(* Logix 5000 project; controller RetoFinal Emulate 5570 rev 30.12; software revision 30.00 *)

TASK MainTask (continuous, watchdog 500 ms) : MainProgram

MODULES
   Local : Emulate 5570 (ICP 2, rev 30.12)
END_MODULES

VAR_GLOBAL   (* controller tags *)
   CajaLlego2 : BOOL;
   CajaPaso2 : BOOL;
   CajaPaso3 : BOOL;
   CondicionInicial : BOOL;
   ControlBarrera : BOOL;
   CounterCajas : COUNTER := (PRE := 1);
   GD_A00 : BOOL;
   GD_A00B : BOOL;
   GD_A01 : BOOL;
   GD_A01B : BOOL;
   GD_A10 : BOOL;
   GD_A10B : BOOL;
   GD_A11 : BOOL;
   GD_A11B : BOOL;
   GD_B0 : BOOL := 1;
   GD_B1 : BOOL;
   GD_B1B : BOOL;
   GD_B2 : BOOL;
   GD_B2B : BOOL;
   GD_B3 : BOOL;
   GD_B3B : BOOL;
   GD_B3C : BOOL;
   GD_B3D : BOOL;
   GD_B4 : BOOL := 1;
   GD_B4B : BOOL := 1;
   GD_B5 : BOOL := 1;
   GD_IN_1 : BOOL;
   GD_IN_2 : BOOL;
   GD_IN_3 : BOOL;
   GD_IN_5 : BOOL;
   GD_IN_6 : BOOL;
   GD_OUT_0 : BOOL;
   GD_OUT_4 : BOOL;
   GD_OUT_5 : BOOL;
   GD_P0 : INT;
   GD_P1 : INT;
   GD_P2 : INT;
   GD_P3 : INT;
   GD_P4 : INT;
   GD_P5 : INT;
   GD_P6 : INT;
   GD_P7 : INT;
   GD_P8 : INT;
   GD_P9 : INT;
   GD_R00 : BOOL := 1;
   GD_R00B : BOOL := 1;
   GD_R01 : BOOL;
   GD_R01B : BOOL;
   GD_R10 : BOOL := 1;
   GD_R11 : BOOL;
   GD_S0 : BOOL;
   GD_S1 : BOOL;
   GD_S10 : BOOL;
   GD_S11 : BOOL;
   GD_S2 : BOOL;
   GD_S3 : BOOL;
   GD_S4 : BOOL;
   GD_S5 : BOOL;
   GD_S6 : BOOL;
   GD_S7 : BOOL;
   GD_S8 : BOOL;
   GD_S9 : BOOL;
   IoT_A00 : BOOL;
   IoT_A01 : BOOL;
   IoT_A10 : BOOL;
   IoT_A11 : BOOL;
   IoT_B0 : BOOL := 1;
   IoT_B1 : BOOL;
   IoT_B2 : BOOL;
   IoT_B3 : BOOL;
   IoT_B4 : BOOL := 1;
   IoT_B5 : BOOL := 1;
   IoT_P0 : INT;
   IoT_P1 : INT;
   IoT_P2 : INT;
   IoT_P3 : INT;
   IoT_P4 : INT;
   IoT_P5 : INT;
   IoT_P6 : INT;
   IoT_P7 : INT;
   IoT_P8 : INT;
   IoT_P9 : INT;
   IoT_R00 : BOOL := 1;
   IoT_R01 : BOOL;
   IoT_R10 : BOOL := 1;
   IoT_R11 : BOOL;
   IoT_S0 : BOOL;
   IoT_S1 : BOOL;
   IoT_S2 : BOOL;
   IoT_S3 : BOOL;
   IoT_S4 : BOOL;
   IoT_S5 : BOOL;
   IoT_S6 : BOOL;
   IoT_S7 : BOOL;
   IoT_S8 : BOOL;
   IoT_S9 : BOOL;
   IoT_Tipo : BOOL;
   Sensor2Down : BOOL;
   Sensor2Up : BOOL;
   Sensor3Up : BOOL;
   T1 : TIMER := (PRE := 1000);
END_VAR

PROGRAM MainProgram   (* main routine MainRoutine *)
VAR
   A00 : BOOL;
   A01 : BOOL;
   A10 : BOOL;
   A11 : BOOL;
   AcomodadorSalidaD : BOOL;
   AcomodadorSalidaL : BOOL;
   B0 : BOOL := 1;
   B1 : BOOL;
   B2 : BOOL;
   B3 : BOOL;
   B4 : BOOL := 1;
   B5 : BOOL := 1;
   C1 : COUNTER := (PRE := 2);
   C2 : COUNTER := (PRE := 2);
   CAJAS : DINT;
   CambioTipo : BOOL;
   E00 : BOOL := 1;
   E001 : BOOL := 1;
   E002 : BOOL;
   E01 : BOOL;
   E1 : BOOL := 1;
   E11 : BOOL := 1;
   E12 : BOOL;
   E2 : BOOL;
   E21 : BOOL;
   E22 : BOOL;
   E23 : BOOL;
   E24 : BOOL;
   E25 : BOOL;
   E26 : BOOL;
   E3 : BOOL := 1;
   F : BOOL;
   F1 : BOOL;
   FIN : BOOL := 1;
   FINE2 : BOOL;
   FINE3 : BOOL;
   GD_IN_4 : BOOL;
   M : BOOL;
   M1 : BOOL;
   P0 : INT;
   P1 : INT;
   P2 : INT;
   P3 : INT;
   P4 : INT;
   P5 : INT;
   P6 : INT;
   P7 : INT;
   P8 : INT;
   P9 : INT;
   R00 : BOOL := 1;
   R01 : BOOL;
   R10 : BOOL := 1;
   R11 : BOOL;
   S0 : BOOL;
   S0D : BOOL;
   S0Dw : BOOL;
   S0U : BOOL;
   S0Up : BOOL;
   S1 : BOOL;
   S10 : BOOL;
   S10D : BOOL;
   S10Dw : BOOL;
   S10U : BOOL;
   S10Up : BOOL;
   S11 : BOOL;
   S11D : BOOL;
   S11Dw : BOOL;
   S11U : BOOL;
   S11Up : BOOL;
   S1D : BOOL;
   S1Dw : BOOL;
   S1U : BOOL;
   S1Up : BOOL;
   S2 : BOOL;
   S2D : BOOL;
   S2Dw : BOOL;
   S2U : BOOL;
   S2Up : BOOL;
   S3 : BOOL;
   S3D : BOOL;
   S3Dw : BOOL;
   S3U : BOOL;
   S3Up : BOOL;
   S4 : BOOL;
   S4D : BOOL;
   S4Dw : BOOL;
   S4U : BOOL;
   S4Up : BOOL;
   S5 : BOOL;
   S5D : BOOL;
   S5Dw : BOOL;
   S5U : BOOL;
   S5Up : BOOL;
   S6 : BOOL;
   S6D : BOOL;
   S6Dw : BOOL;
   S6U : BOOL;
   S6Up : BOOL;
   S7 : BOOL;
   S7D : BOOL;
   S7Dw : BOOL;
   S7U : BOOL;
   S7Up : BOOL;
   S8 : BOOL;
   S8D : BOOL;
   S8Dw : BOOL;
   S8U : BOOL;
   S8Up : BOOL;
   S9 : BOOL;
   S9D : BOOL;
   S9Dw : BOOL;
   S9U : BOOL;
   S9Up : BOOL;
   SistemaActivo : BOOL := 1;
   TimerBarrera : TIMER := (PRE := 500);
   Tipo : BOOL;
   TipoD : BOOL;
   TipoDw : BOOL;
   TipoU : BOOL;
   TipoUp : BOOL;
END_VAR

ROUTINE A   (* ladder *)
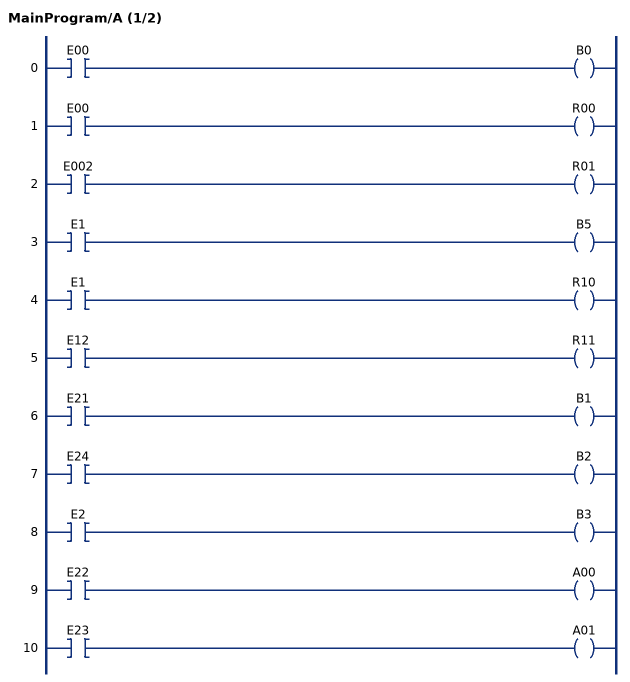
   0: XIC(E00)OTE(B0);
   1: XIC(E00)OTE(R00);
   2: XIC(E002)OTE(R01);
   3: XIC(E1)OTE(B5);
   4: XIC(E1)OTE(R10);
   5: XIC(E12)OTE(R11);
   6: XIC(E21)OTE(B1);
   7: XIC(E24)OTE(B2);
   8: XIC(E2)OTE(B3);
   9: XIC(E22)OTE(A00);
   10: XIC(E23)OTE(A01);
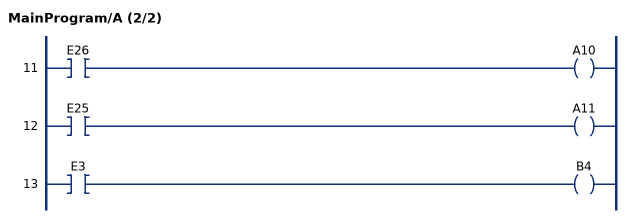
   11: XIC(E26)OTE(A10);
   12: XIC(E25)OTE(A11);
   13: XIC(E3)OTE(B4);
END_ROUTINE

ROUTINE Buffer   (* ladder *)
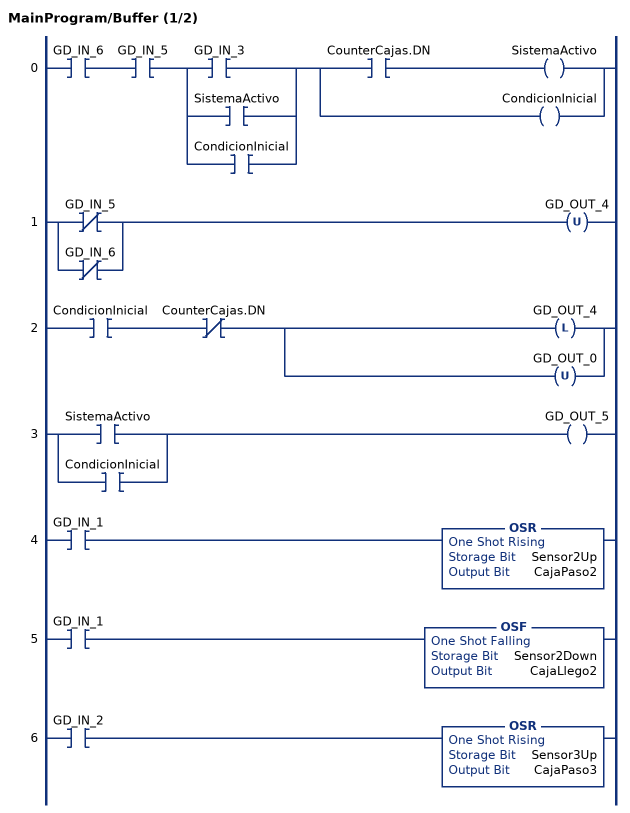
   0: XIC(GD_IN_6)XIC(GD_IN_5)[XIC(GD_IN_3) ,[XIC(SistemaActivo) ,XIC(CondicionInicial) ] ][XIC(CounterCajas.DN) OTE(SistemaActivo) ,OTE(CondicionInicial) ];
   1: [XIO(GD_IN_5) ,XIO(GD_IN_6) ]OTU(GD_OUT_4);
   2: XIC(CondicionInicial)XIO(CounterCajas.DN)[OTL(GD_OUT_4) ,OTU(GD_OUT_0) ];
   3: [XIC(SistemaActivo) ,XIC(CondicionInicial) ]OTE(GD_OUT_5);
   4: XIC(GD_IN_1)OSR(Sensor2Up,CajaPaso2);
   5: XIC(GD_IN_1)OSF(Sensor2Down,CajaLlego2);
   6: XIC(GD_IN_2)OSR(Sensor3Up,CajaPaso3);
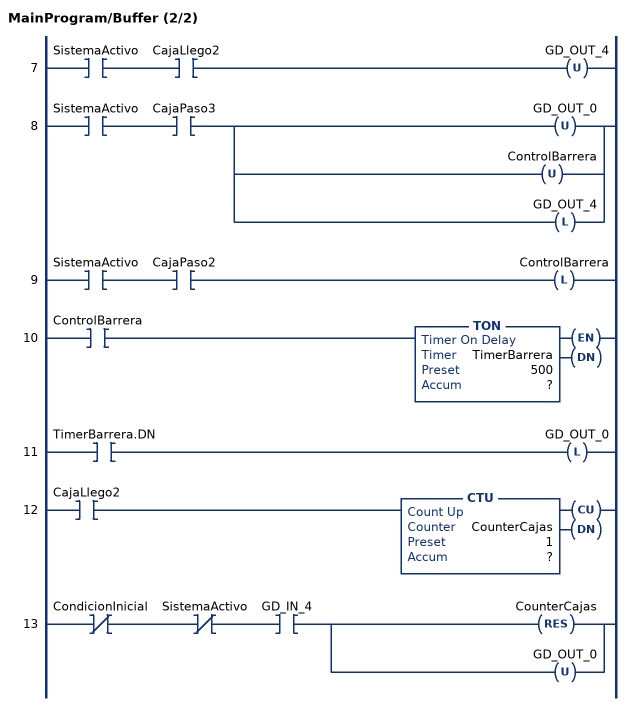
   7: XIC(SistemaActivo)XIC(CajaLlego2)OTU(GD_OUT_4);
   8: XIC(SistemaActivo)XIC(CajaPaso3)[OTU(GD_OUT_0) ,[OTU(ControlBarrera) ,OTL(GD_OUT_4) ] ];
   9: XIC(SistemaActivo)XIC(CajaPaso2)OTL(ControlBarrera);
   10: XIC(ControlBarrera)TON(TimerBarrera,?,?);
   11: XIC(TimerBarrera.DN)OTL(GD_OUT_0);
   12: XIC(CajaLlego2)CTU(CounterCajas,?,?);
   13: XIO(CondicionInicial)XIO(SistemaActivo)XIC(GD_IN_4)[RES(CounterCajas) ,OTU(GD_OUT_0) ];
END_ROUTINE

ROUTINE C   (* ladder *)
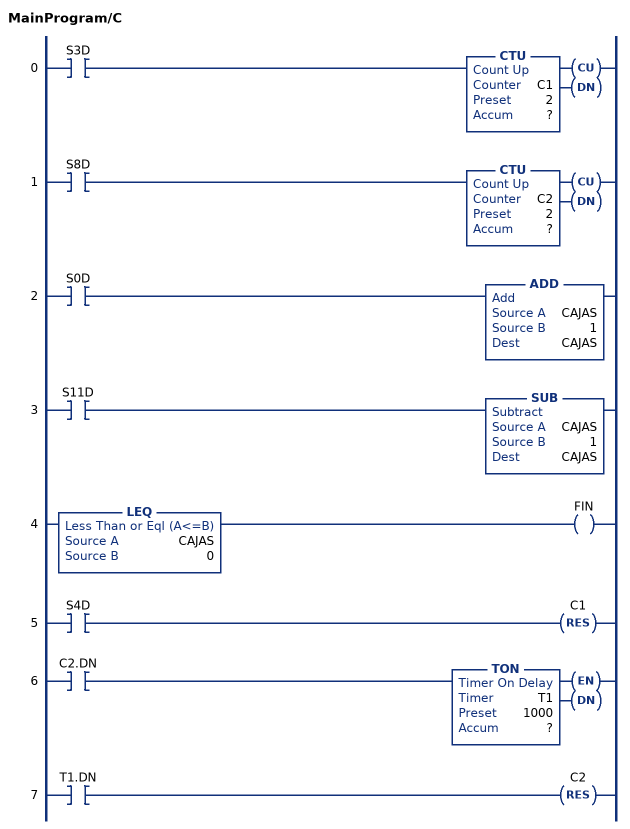
   0: XIC(S3D)CTU(C1,?,?);
   1: XIC(S8D)CTU(C2,?,?);
   2: XIC(S0D)ADD(CAJAS,1,CAJAS);
   3: XIC(S11D)SUB(CAJAS,1,CAJAS);
   4: LEQ(CAJAS,0)OTE(FIN);
   5: XIC(S4D)RES(C1);
   6: XIC(C2.DN)TON(T1,?,?);
   7: XIC(T1.DN)RES(C2);
END_ROUTINE

ROUTINE E   (* ladder *)
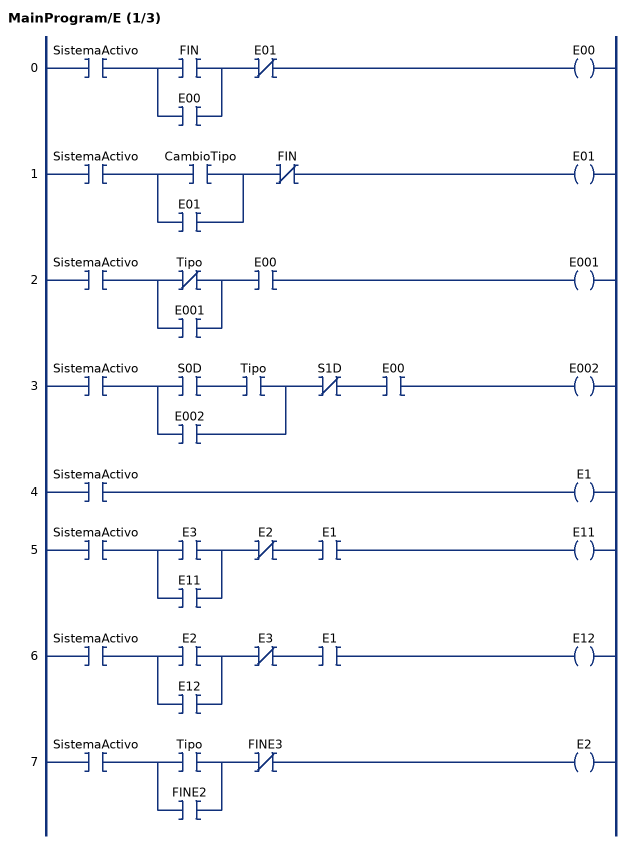
   0: XIC(SistemaActivo)[XIC(FIN) ,XIC(E00) ]XIO(E01)OTE(E00);
   1: XIC(SistemaActivo)[XIC(CambioTipo) ,XIC(E01) ]XIO(FIN)OTE(E01);
   2: XIC(SistemaActivo)[XIO(Tipo) ,XIC(E001) ]XIC(E00)OTE(E001);
   3: XIC(SistemaActivo)[XIC(S0D) XIC(Tipo) ,XIC(E002) ]XIO(S1D)XIC(E00)OTE(E002);
   4: XIC(SistemaActivo)OTE(E1);
   5: XIC(SistemaActivo)[XIC(E3) ,XIC(E11) ]XIO(E2)XIC(E1)OTE(E11);
   6: XIC(SistemaActivo)[XIC(E2) ,XIC(E12) ]XIO(E3)XIC(E1)OTE(E12);
   7: XIC(SistemaActivo)[XIC(Tipo) ,XIC(FINE2) ]XIO(FINE3)OTE(E2);
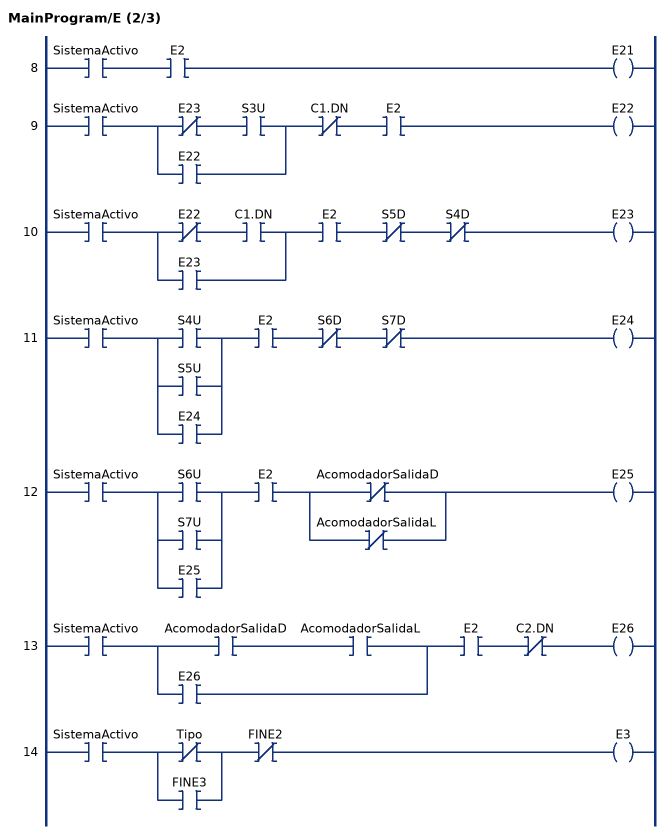
   8: XIC(SistemaActivo)XIC(E2)OTE(E21);
   9: XIC(SistemaActivo)[XIO(E23) XIC(S3U) ,XIC(E22) ]XIO(C1.DN)XIC(E2)OTE(E22);
   10: XIC(SistemaActivo)[XIO(E22) XIC(C1.DN) ,XIC(E23) ]XIC(E2)XIO(S5D)XIO(S4D)OTE(E23);
   11: XIC(SistemaActivo)[[XIC(S4U) ,XIC(S5U) ] ,XIC(E24) ]XIC(E2)XIO(S6D)XIO(S7D)OTE(E24);
   12: XIC(SistemaActivo)[[XIC(S6U) ,XIC(S7U) ] ,XIC(E25) ]XIC(E2)[XIO(AcomodadorSalidaD) ,XIO(AcomodadorSalidaL) ]OTE(E25);
   13: XIC(SistemaActivo)[XIC(AcomodadorSalidaD) XIC(AcomodadorSalidaL) ,XIC(E26) ]XIC(E2)XIO(C2.DN)OTE(E26);
   14: XIC(SistemaActivo)[XIO(Tipo) ,XIC(FINE3) ]XIO(FINE2)OTE(E3);
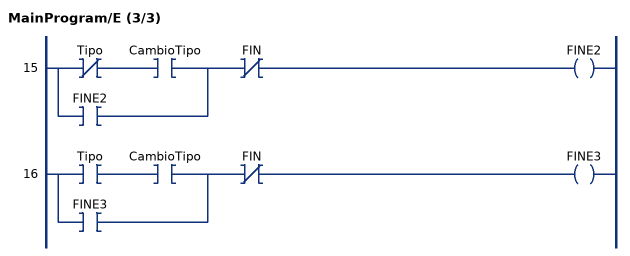
   15: [XIO(Tipo) XIC(CambioTipo) ,XIC(FINE2) ]XIO(FIN)OTE(FINE2);
   16: [XIC(Tipo) XIC(CambioTipo) ,XIC(FINE3) ]XIO(FIN)OTE(FINE3);
END_ROUTINE

ROUTINE GD   (* ladder *)
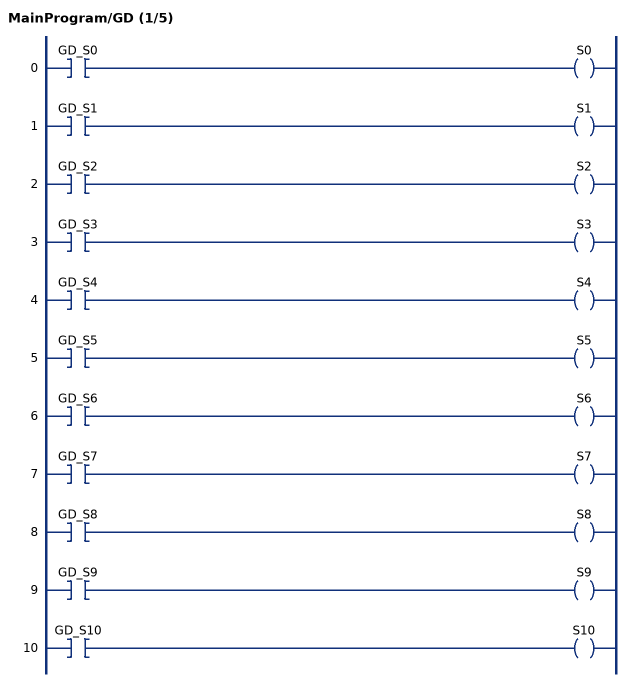
   0: XIC(GD_S0)OTE(S0);
   1: XIC(GD_S1)OTE(S1);
   2: XIC(GD_S2)OTE(S2);
   3: XIC(GD_S3)OTE(S3);
   4: XIC(GD_S4)OTE(S4);
   5: XIC(GD_S5)OTE(S5);
   6: XIC(GD_S6)OTE(S6);
   7: XIC(GD_S7)OTE(S7);
   8: XIC(GD_S8)OTE(S8);
   9: XIC(GD_S9)OTE(S9);
   10: XIC(GD_S10)OTE(S10);
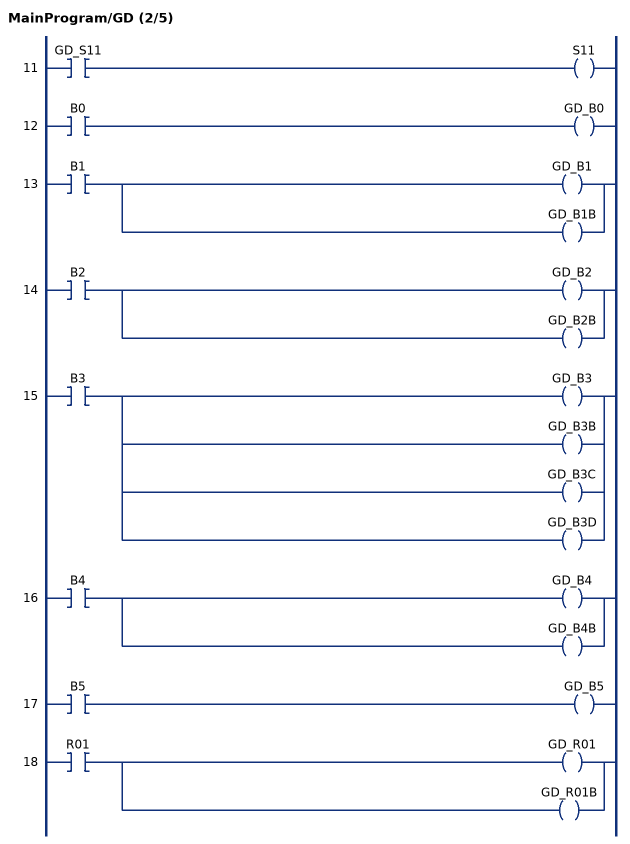
   11: XIC(GD_S11)OTE(S11);
   12: XIC(B0)OTE(GD_B0);
   13: XIC(B1)[OTE(GD_B1) ,OTE(GD_B1B) ];
   14: XIC(B2)[OTE(GD_B2) ,OTE(GD_B2B) ];
   15: XIC(B3)[OTE(GD_B3) ,[OTE(GD_B3B) ,[OTE(GD_B3C) ,OTE(GD_B3D) ] ] ];
   16: XIC(B4)[OTE(GD_B4) ,OTE(GD_B4B) ];
   17: XIC(B5)OTE(GD_B5);
   18: XIC(R01)[OTE(GD_R01) ,OTE(GD_R01B) ];
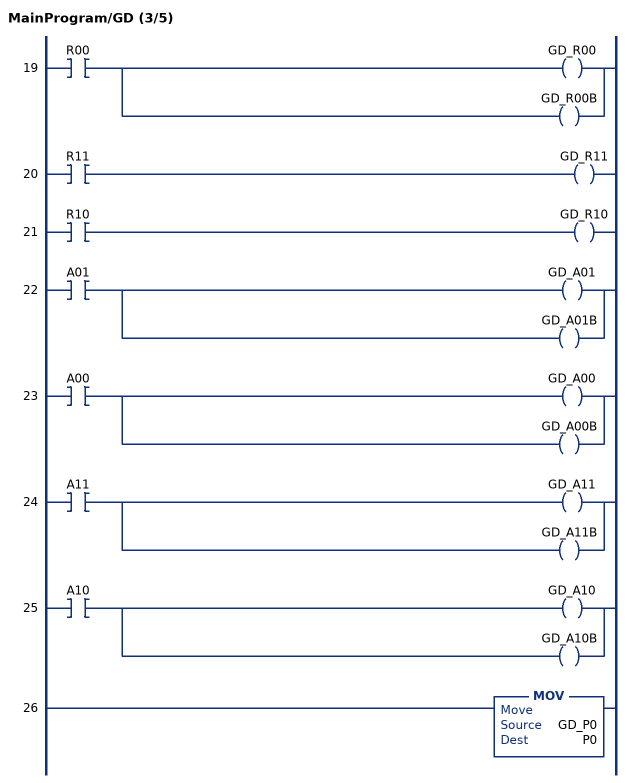
   19: XIC(R00)[OTE(GD_R00) ,OTE(GD_R00B) ];
   20: XIC(R11)OTE(GD_R11);
   21: XIC(R10)OTE(GD_R10);
   22: XIC(A01)[OTE(GD_A01) ,OTE(GD_A01B) ];
   23: XIC(A00)[OTE(GD_A00) ,OTE(GD_A00B) ];
   24: XIC(A11)[OTE(GD_A11) ,OTE(GD_A11B) ];
   25: XIC(A10)[OTE(GD_A10) ,OTE(GD_A10B) ];
   26: MOV(GD_P0,P0);
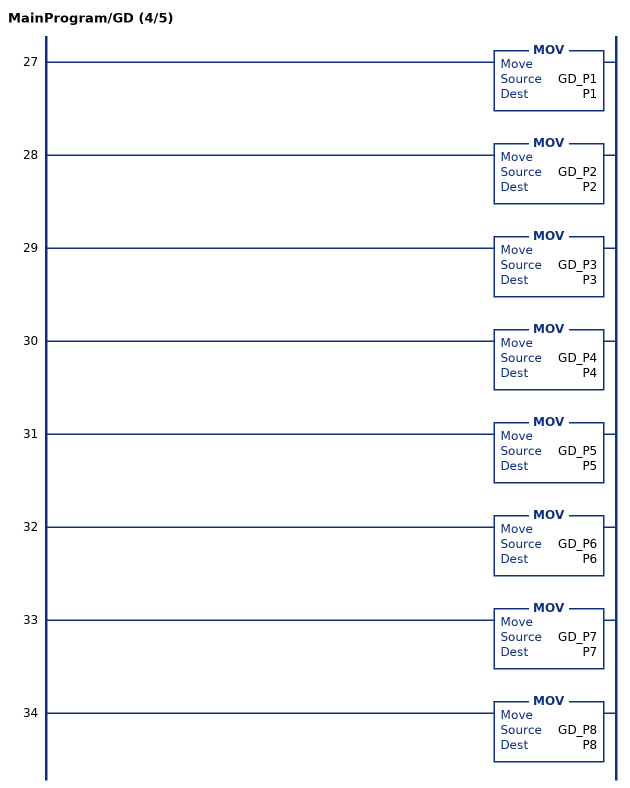
   27: MOV(GD_P1,P1);
   28: MOV(GD_P2,P2);
   29: MOV(GD_P3,P3);
   30: MOV(GD_P4,P4);
   31: MOV(GD_P5,P5);
   32: MOV(GD_P6,P6);
   33: MOV(GD_P7,P7);
   34: MOV(GD_P8,P8);
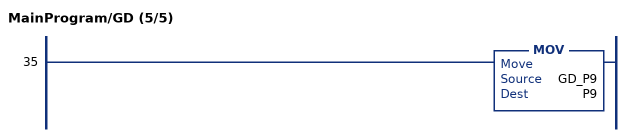
   35: MOV(GD_P9,P9);
END_ROUTINE

ROUTINE IoT   (* ladder *)
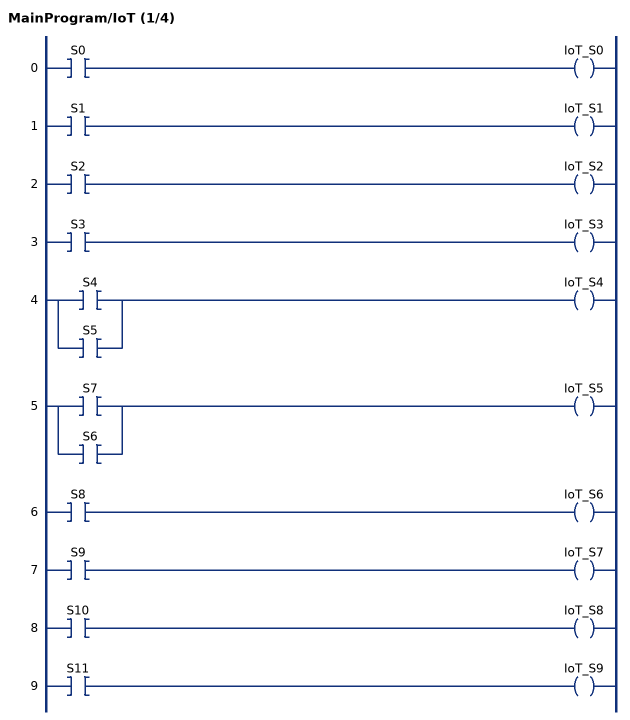
   0: XIC(S0)OTE(IoT_S0);
   1: XIC(S1)OTE(IoT_S1);
   2: XIC(S2)OTE(IoT_S2);
   3: XIC(S3)OTE(IoT_S3);
   4: [XIC(S4) ,XIC(S5) ]OTE(IoT_S4);
   5: [XIC(S7) ,XIC(S6) ]OTE(IoT_S5);
   6: XIC(S8)OTE(IoT_S6);
   7: XIC(S9)OTE(IoT_S7);
   8: XIC(S10)OTE(IoT_S8);
   9: XIC(S11)OTE(IoT_S9);
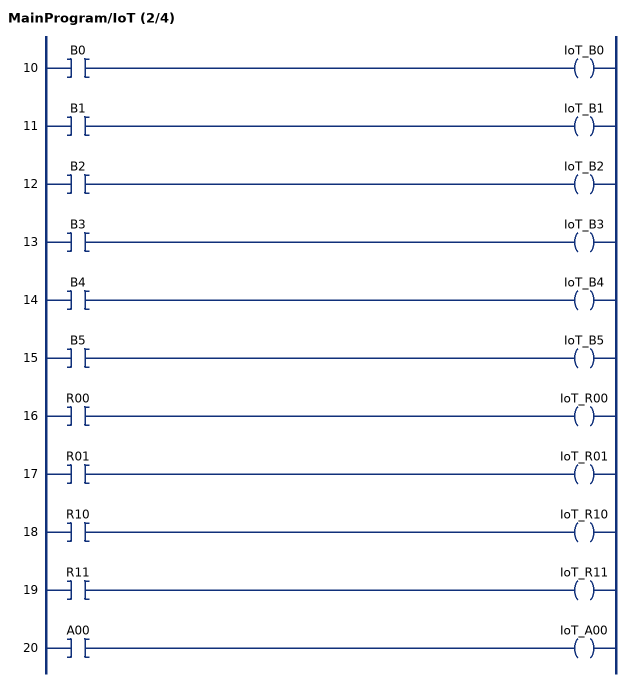
   10: XIC(B0)OTE(IoT_B0);
   11: XIC(B1)OTE(IoT_B1);
   12: XIC(B2)OTE(IoT_B2);
   13: XIC(B3)OTE(IoT_B3);
   14: XIC(B4)OTE(IoT_B4);
   15: XIC(B5)OTE(IoT_B5);
   16: XIC(R00)OTE(IoT_R00);
   17: XIC(R01)OTE(IoT_R01);
   18: XIC(R10)OTE(IoT_R10);
   19: XIC(R11)OTE(IoT_R11);
   20: XIC(A00)OTE(IoT_A00);
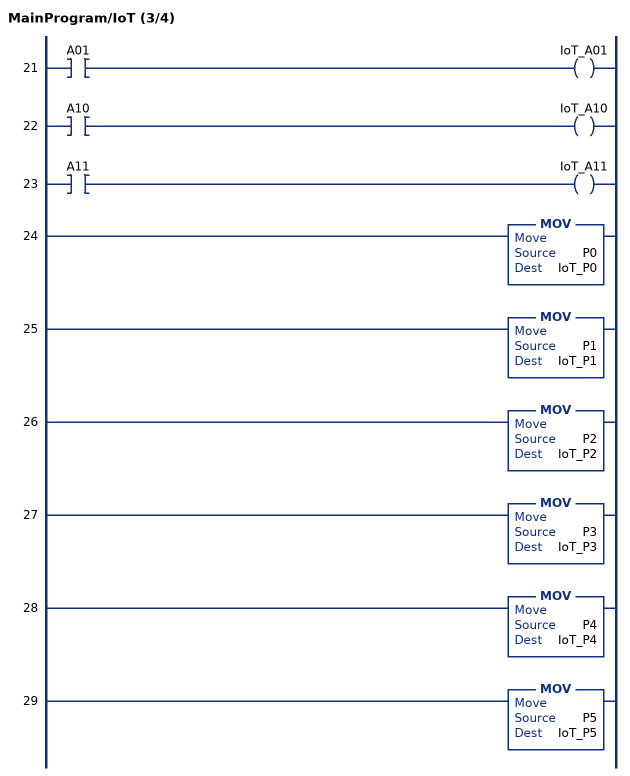
   21: XIC(A01)OTE(IoT_A01);
   22: XIC(A10)OTE(IoT_A10);
   23: XIC(A11)OTE(IoT_A11);
   24: MOV(P0,IoT_P0);
   25: MOV(P1,IoT_P1);
   26: MOV(P2,IoT_P2);
   27: MOV(P3,IoT_P3);
   28: MOV(P4,IoT_P4);
   29: MOV(P5,IoT_P5);
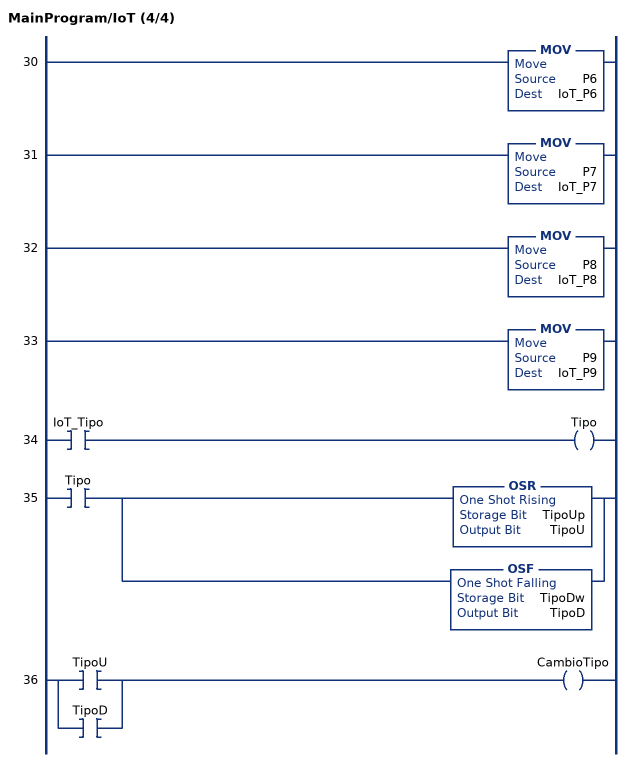
   30: MOV(P6,IoT_P6);
   31: MOV(P7,IoT_P7);
   32: MOV(P8,IoT_P8);
   33: MOV(P9,IoT_P9);
   34: XIC(IoT_Tipo)OTE(Tipo);
   35: XIC(Tipo)[OSR(TipoUp,TipoU) ,OSF(TipoDw,TipoD) ];
   36: [XIC(TipoU) ,XIC(TipoD) ]OTE(CambioTipo);
END_ROUTINE

ROUTINE MainRoutine   (* ladder *)
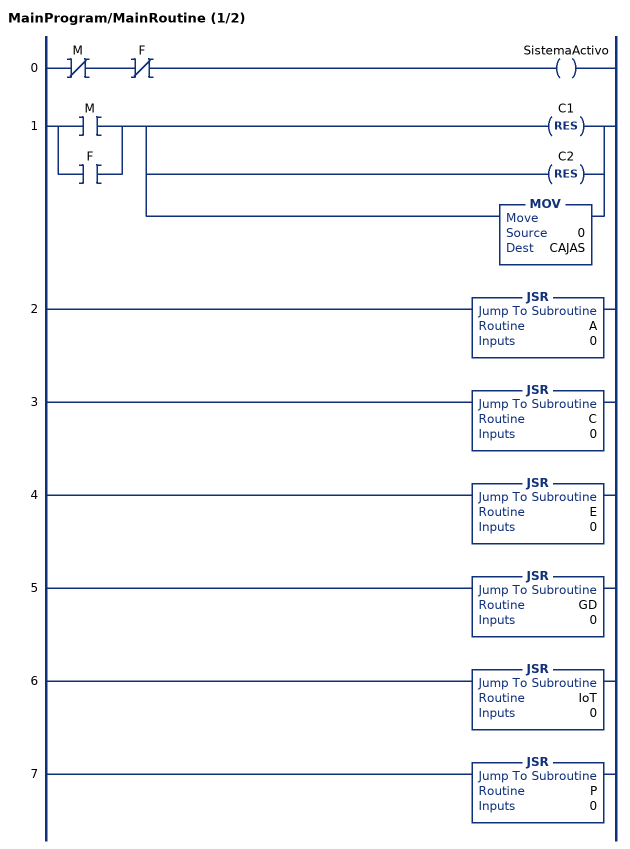
   0: XIO(M)XIO(F)OTE(SistemaActivo);
   1: [XIC(M) ,XIC(F) ][RES(C1) ,[RES(C2) ,MOV(0,CAJAS) ] ];
   2: JSR(A,0);
   3: JSR(C,0);
   4: JSR(E,0);
   5: JSR(GD,0);
   6: JSR(IoT,0);
   7: JSR(P,0);
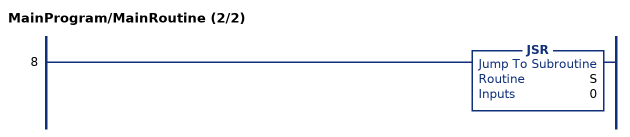
   8: JSR(S,0);
END_ROUTINE

ROUTINE P   (* ladder *)
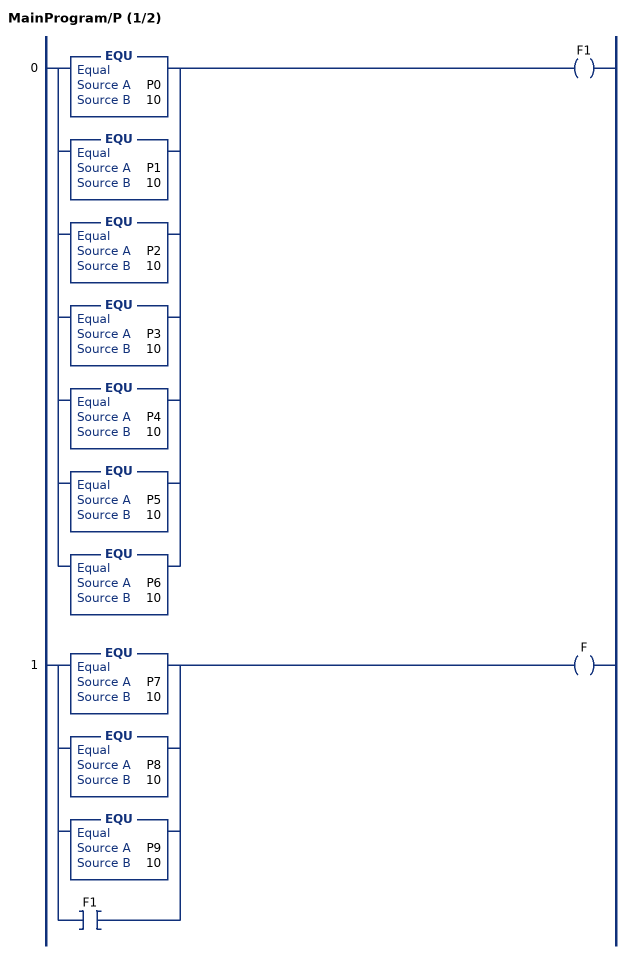
   0: [EQU(P0,10) ,[EQU(P1,10) ,[EQU(P2,10) ,[EQU(P3,10) ,[EQU(P4,10) ,[EQU(P5,10) ,EQU(P6,10) ] ] ] ] ] ]OTE(F1);
   1: [EQU(P7,10) ,[EQU(P8,10) ,[EQU(P9,10) ,XIC(F1) ] ] ]OTE(F);
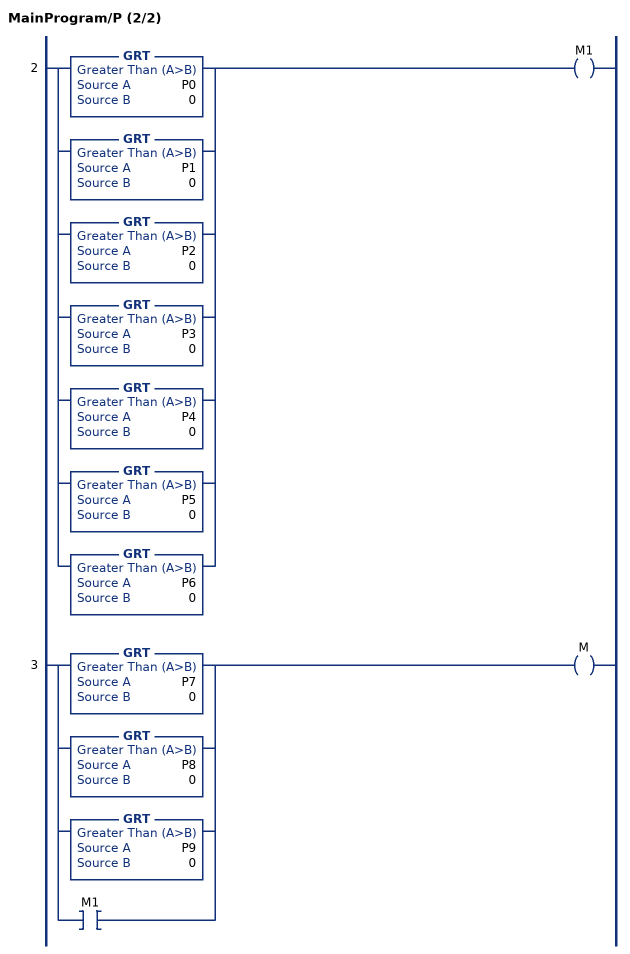
   2: [GRT(P0,0) ,[GRT(P1,0) ,[GRT(P2,0) ,[GRT(P3,0) ,[GRT(P4,0) ,[GRT(P5,0) ,GRT(P6,0) ] ] ] ] ] ]OTE(M1);
   3: [GRT(P7,0) ,[GRT(P8,0) ,[GRT(P9,0) ,XIC(M1) ] ] ]OTE(M);
END_ROUTINE

ROUTINE S   (* ladder *)
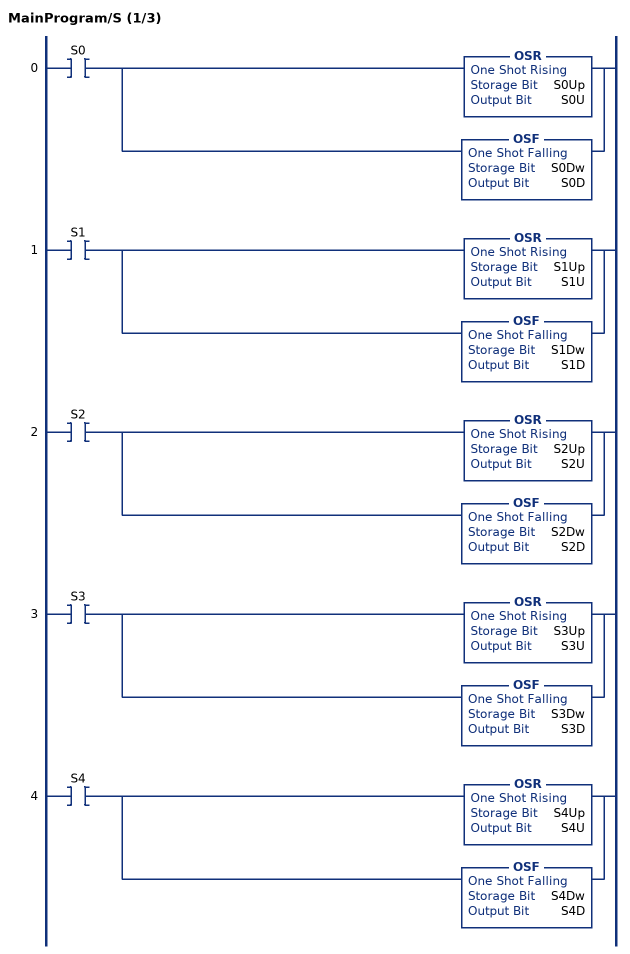
   0: XIC(S0)[OSR(S0Up,S0U) ,OSF(S0Dw,S0D) ];
   1: XIC(S1)[OSR(S1Up,S1U) ,OSF(S1Dw,S1D) ];
   2: XIC(S2)[OSR(S2Up,S2U) ,OSF(S2Dw,S2D) ];
   3: XIC(S3)[OSR(S3Up,S3U) ,OSF(S3Dw,S3D) ];
   4: XIC(S4)[OSR(S4Up,S4U) ,OSF(S4Dw,S4D) ];
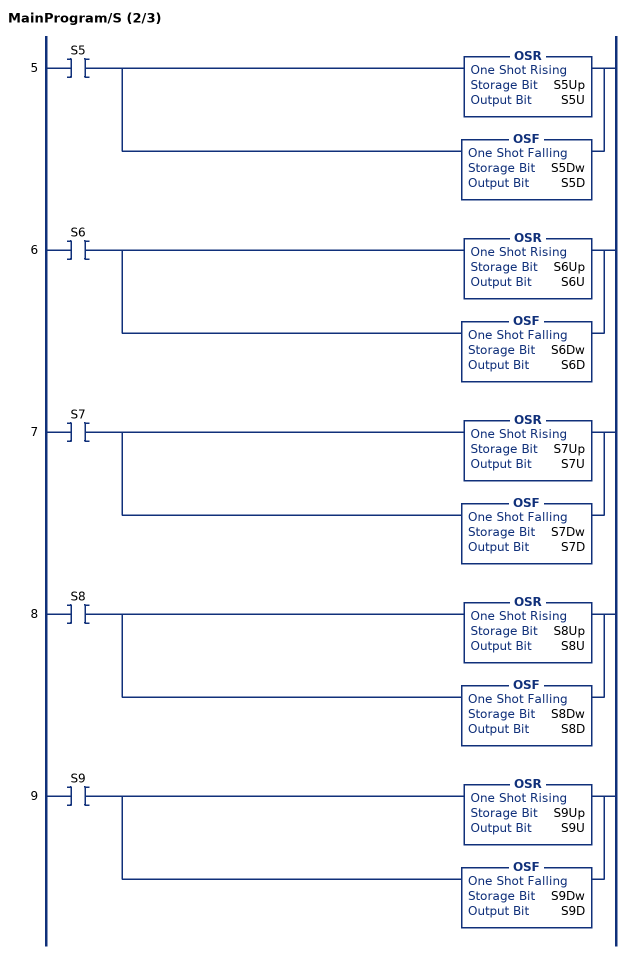
   5: XIC(S5)[OSR(S5Up,S5U) ,OSF(S5Dw,S5D) ];
   6: XIC(S6)[OSR(S6Up,S6U) ,OSF(S6Dw,S6D) ];
   7: XIC(S7)[OSR(S7Up,S7U) ,OSF(S7Dw,S7D) ];
   8: XIC(S8)[OSR(S8Up,S8U) ,OSF(S8Dw,S8D) ];
   9: XIC(S9)[OSR(S9Up,S9U) ,OSF(S9Dw,S9D) ];
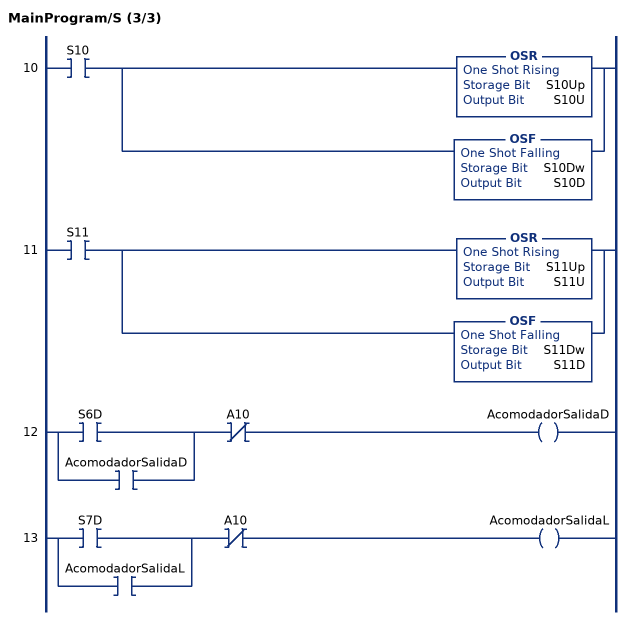
   10: XIC(S10)[OSR(S10Up,S10U) ,OSF(S10Dw,S10D) ];
   11: XIC(S11)[OSR(S11Up,S11U) ,OSF(S11Dw,S11D) ];
   12: [XIC(S6D) ,XIC(AcomodadorSalidaD) ]XIO(A10)OTE(AcomodadorSalidaD);
   13: [XIC(S7D) ,XIC(AcomodadorSalidaL) ]XIO(A10)OTE(AcomodadorSalidaL);
END_ROUTINE
END_PROGRAM
